// Check total duration of profiles
AssertEquals_LREAL(Expected := 4.0, Actual := ruckig.Trajectory.Duration, DELTA := 1E-8, Message := 'Duration incorrect');

// Check minimum duration
AssertEquals_LREAL(Expected := input.MinDuration, Actual := ruckig.Trajectory.Duration, DELTA := 1E-8, Message := 'Minimum duration not equals duration');

// Check duration for each phase
positionExtrema := ruckig.Trajectory._profiles[0].positionExtrema();
AssertEquals_LREAL(0.0, positionExtrema.Tmax, 1E-9, message:='Profile[0] Tmax incorrect');
AssertEquals_LREAL(61.37396011937787, positionExtrema.Maximum, 1E-9, message:='Profile[0] maximum incorrect');
AssertEquals_LREAL(4.0, positionExtrema.Tmin, 1E-9, message:='Profile[0] Tmin incorrect');
AssertEquals_LREAL(-932.2714554581783, positionExtrema.Minimum, 1E-9, message:='Profile[0] minimum incorrect');

positionExtrema := ruckig.Trajectory._profiles[1].positionExtrema();
AssertEquals_LREAL(4.0, positionExtrema.Tmax, 1E-9, message:='Profile[1] Tmax incorrect');
AssertEquals_LREAL(3356.191464991089, positionExtrema.Maximum, 1E-9, message:='Profile[1] maximum incorrect');
AssertEquals_LREAL(0.10412338784096734, positionExtrema.Tmin, 1E-9, message:='Profile[1] Tmin incorrect');
AssertEquals_LREAL(68.24379604148844, positionExtrema.Minimum, 1E-9, message:='Profile[1] minimum incorrect');

positionExtrema := ruckig.Trajectory._profiles[2].positionExtrema();
AssertEquals_LREAL(0.0, positionExtrema.Tmax, 1E-9, message:='Profile[2] Tmax incorrect');
AssertEquals_LREAL(-8.257039659155268, positionExtrema.Maximum, 1E-9, message:='Profile[2] maximum incorrect');
AssertEquals_LREAL(4.0, positionExtrema.Tmin, 1E-9, message:='Profile[2] Tmin incorrect');
AssertEquals_LREAL(-2142.4383401030323, positionExtrema.Minimum, 1E-9, message:='Profile[2] minimum incorrect');
   

TEST_FINISHED();
END_METHOD

METHOD Test_Trajectory_VelIntrf_HasMinDuration_HasTargetVelocity_HasTargetAcceleration_25
VAR_INST
  ruckig : Struckig.Ruckig(0.001, 0);
  input : Struckig.InputParameter(3) := (
    ControlInterface := ControlInterfaceType.Velocity,
    Synchronization := SynchronizationType.TimeSync,
    MinDuration := 5.0,
    MaxVelocity := [ 2000.0, 2000.0, 2000.0 ],
    MaxAcceleration := [ 20000.0, 20000.0, 20000.0 ],
    MaxJerk := [ 800000.0, 800000.0, 800000.0 ],
    CurrentPosition := [ 99.27158709173054, 51.78630599017913, -82.71240030046118 ],
    CurrentVelocity := [ 617.0096879713556, 556.3356400770322, 654.4714219366203 ],
    CurrentAcceleration := [ 574.9072883020708, 8161.605381343747, 7215.343607485673 ],
    TargetPosition := [ -75.73302485201327, -76.60258111111662, -93.84383456920497 ],
    TargetVelocity := [ -134.5020942775601, 636.5230467842334, -659.8475456020238 ],
    TargetAcceleration := [ -262.53891173287866, -851.053910299499, -307.5361794862756 ]
  );
  
  positionExtrema : Struckig.PositionExtremaDesc;
END_VAR
TEST('Trajectory_VelIntrf_HasMinDuration_HasTargetVelocity_HasTargetAcceleration_25');

ruckig(Input:=input);

// Check total duration of profiles
AssertEquals_LREAL(Expected := 5.0, Actual := ruckig.Trajectory.Duration, DELTA := 1E-8, Message := 'Duration incorrect');

// Check minimum duration
AssertEquals_LREAL(Expected := input.MinDuration, Actual := ruckig.Trajectory.Duration, DELTA := 1E-8, Message := 'Minimum duration not equals duration');

// Check duration for each phase
positionExtrema := ruckig.Trajectory._profiles[0].positionExtrema();
AssertEquals_LREAL(5.0, positionExtrema.Tmax, 1E-9, message:='Profile[0] Tmax incorrect');
AssertEquals_LREAL(2457.793957890017, positionExtrema.Maximum, 1E-9, message:='Profile[0] maximum incorrect');
AssertEquals_LREAL(0.0, positionExtrema.Tmin, 1E-9, message:='Profile[0] Tmin incorrect');
AssertEquals_LREAL(99.27158709173054, positionExtrema.Minimum, 1E-9, message:='Profile[0] minimum incorrect');

positionExtrema := ruckig.Trajectory._profiles[1].positionExtrema();
AssertEquals_LREAL(5.0, positionExtrema.Tmax, 1E-9, message:='Profile[1] Tmax incorrect');
AssertEquals_LREAL(12482.220923700503, positionExtrema.Maximum, 1E-9, message:='Profile[1] maximum incorrect');
AssertEquals_LREAL(0.0, positionExtrema.Tmin, 1E-9, message:='Profile[1] Tmin incorrect');
AssertEquals_LREAL(51.78630599017913, positionExtrema.Minimum, 1E-9, message:='Profile[1] minimum incorrect');

positionExtrema := ruckig.Trajectory._profiles[2].positionExtrema();
AssertEquals_LREAL(5.0, positionExtrema.Tmax, 1E-9, message:='Profile[2] Tmax incorrect');
AssertEquals_LREAL(457.83088712667626, positionExtrema.Maximum, 1E-9, message:='Profile[2] maximum incorrect');
AssertEquals_LREAL(0.0, positionExtrema.Tmin, 1E-9, message:='Profile[2] Tmin incorrect');
AssertEquals_LREAL(-82.71240030046118, positionExtrema.Minimum, 1E-9, message:='Profile[2] minimum incorrect');
   

TEST_FINISHED();
END_METHOD

METHOD Test_Trajectory_VelIntrf_HasMinDuration_HasTargetVelocity_HasTargetAcceleration_26
VAR_INST
  ruckig : Struckig.Ruckig(0.001, 0);
  input : Struckig.InputParameter(3) := (
    ControlInterface := ControlInterfaceType.Velocity,
    Synchronization := SynchronizationType.TimeSync,
    MinDuration := 2.0,
    MaxVelocity := [ 2000.0, 2000.0, 2000.0 ],
    MaxAcceleration := [ 20000.0, 20000.0, 20000.0 ],
    MaxJerk := [ 800000.0, 800000.0, 800000.0 ],
    CurrentPosition := [ 47.83664173753348, -4.090200694219973, 75.62715399288581 ],
    CurrentVelocity := [ -412.71660212910535, -344.97977752529744, -662.3972561668236 ],
    CurrentAcceleration := [ 9700.323608694027, 4925.451680171778, 528.779511900253 ],
    TargetPosition := [ -26.350792724711255, -10.804969468053471, -80.84927076896919 ],
    TargetVelocity := [ -661.2515009925905, -544.0751045990595, 389.8586138148876 ],
    TargetAcceleration := [ -326.74185324603604, 477.02942558038353, -127.6960040536186 ]
  );
  
  positionExtrema : Struckig.PositionExtremaDesc;
END_VAR
TEST('Trajectory_VelIntrf_HasMinDuration_HasTargetVelocity_HasTargetAcceleration_26');

ruckig(Input:=input);

// Check total duration of profiles
AssertEquals_LREAL(Expected := 2.0, Actual := ruckig.Trajectory.Duration, DELTA := 1E-8, Message := 'Duration incorrect');

// Check minimum duration
AssertEquals_LREAL(Expected := input.MinDuration, Actual := ruckig.Trajectory.Duration, DELTA := 1E-8, Message := 'Minimum duration not equals duration');

// Check duration for each phase
positionExtrema := ruckig.Trajectory._profiles[0].positionExtrema();
AssertEquals_LREAL(0.0, positionExtrema.Tmax, 1E-9, message:='Profile[0] Tmax incorrect');
AssertEquals_LREAL(47.83664173753348, positionExtrema.Maximum, 1E-9, message:='Profile[0] maximum incorrect');
AssertEquals_LREAL(2.0, positionExtrema.Tmin, 1E-9, message:='Profile[0] Tmin incorrect');
AssertEquals_LREAL(-965.6623915281051, positionExtrema.Minimum, 1E-9, message:='Profile[0] minimum incorrect');

positionExtrema := ruckig.Trajectory._profiles[1].positionExtrema();
AssertEquals_LREAL(0.0, positionExtrema.Tmax, 1E-9, message:='Profile[1] Tmax incorrect');
AssertEquals_LREAL(-4.090200694219973, positionExtrema.Maximum, 1E-9, message:='Profile[1] maximum incorrect');
AssertEquals_LREAL(2.0, positionExtrema.Tmin, 1E-9, message:='Profile[1] Tmin incorrect');
AssertEquals_LREAL(-877.5597601233831, positionExtrema.Minimum, 1E-9, message:='Profile[1] minimum incorrect');

positionExtrema := ruckig.Trajectory._profiles[2].positionExtrema();
AssertEquals_LREAL(0.0, positionExtrema.Tmax, 1E-9, message:='Profile[2] Tmax incorrect');
AssertEquals_LREAL(75.62715399288581, positionExtrema.Maximum, 1E-9, message:='Profile[2] maximum incorrect');
AssertEquals_LREAL(1.9991825530237812, positionExtrema.Tmin, 1E-9, message:='Profile[2] Tmin incorrect');
AssertEquals_LREAL(-196.96292798248453, positionExtrema.Minimum, 1E-9, message:='Profile[2] minimum incorrect');
   

TEST_FINISHED();
END_METHOD

METHOD Test_Trajectory_VelIntrf_HasMinDuration_HasTargetVelocity_HasTargetAcceleration_33
VAR_INST
  ruckig : Struckig.Ruckig(0.001, 0);
  input : Struckig.InputParameter(3) := (
    ControlInterface := ControlInterfaceType.Velocity,
    Synchronization := SynchronizationType.TimeSync,
    MinDuration := 1.0,
    MaxVelocity := [ 2000.0, 2000.0, 2000.0 ],
    MaxAcceleration := [ 20000.0, 20000.0, 20000.0 ],
    MaxJerk := [ 800000.0, 800000.0, 800000.0 ],
    CurrentPosition := [ -49.2031444482373, -51.45640574706518, 70.88792157601674 ],
    CurrentVelocity := [ -496.32492650532754, -32.672137553484845, 433.6351152131574 ],
    CurrentAcceleration := [ 5796.767034802937, 149.52817879179565, 5479.773632181257 ],
    TargetPosition := [ -60.683308313785076, -77.36542095799315, 35.25281163323578 ],
    TargetVelocity := [ -239.87671609275264, 822.5237555037947, -341.77342454738846 ],
    TargetAcceleration := [ 442.7287565429956, -997.6913770242959, -816.4447449025389 ]
  );
  
  positionExtrema : Struckig.PositionExtremaDesc;
END_VAR
TEST('Trajectory_VelIntrf_HasMinDuration_HasTargetVelocity_HasTargetAcceleration_33');

ruckig(Input:=input);

// Check total duration of profiles
AssertEquals_LREAL(Expected := 1.0, Actual := ruckig.Trajectory.Duration, DELTA := 1E-8, Message := 'Duration incorrect');

// Check minimum duration
AssertEquals_LREAL(Expected := input.MinDuration, Actual := ruckig.Trajectory.Duration, DELTA := 1E-8, Message := 'Minimum duration not equals duration');

// Check duration for each phase
positionExtrema := ruckig.Trajectory._profiles[0].positionExtrema();
AssertEquals_LREAL(0.0, positionExtrema.Tmax, 1E-9, message:='Profile[0] Tmax incorrect');
AssertEquals_LREAL(-49.2031444482373, positionExtrema.Maximum, 1E-9, message:='Profile[0] maximum incorrect');
AssertEquals_LREAL(1.0, positionExtrema.Tmin, 1E-9, message:='Profile[0] Tmin incorrect');
AssertEquals_LREAL(-407.7025966385173, positionExtrema.Minimum, 1E-9, message:='Profile[0] minimum incorrect');

positionExtrema := ruckig.Trajectory._profiles[1].positionExtrema();
AssertEquals_LREAL(1.0, positionExtrema.Tmax, 1E-9, message:='Profile[1] Tmax incorrect');
AssertEquals_LREAL(344.3868574234848, positionExtrema.Maximum, 1E-9, message:='Profile[1] maximum incorrect');
AssertEquals_LREAL(0.000885165723529272, positionExtrema.Tmin, 1E-9, message:='Profile[1] Tmin incorrect');
AssertEquals_LREAL(-51.485174951826146, positionExtrema.Minimum, 1E-9, message:='Profile[1] minimum incorrect');

positionExtrema := ruckig.Trajectory._profiles[2].positionExtrema();
AssertEquals_LREAL(0.9999795141123666, positionExtrema.Tmax, 1E-9, message:='Profile[2] Tmax incorrect');
AssertEquals_LREAL(129.085190687188, positionExtrema.Maximum, 1E-9, message:='Profile[2] maximum incorrect');
AssertEquals_LREAL(0.0, positionExtrema.Tmin, 1E-9, message:='Profile[2] Tmin incorrect');
AssertEquals_LREAL(70.88792157601674, positionExtrema.Minimum, 1E-9, message:='Profile[2] minimum incorrect');
   

TEST_FINISHED();
END_METHOD

METHOD Test_Trajectory_VelIntrf_HasMinDuration_HasTargetVelocity_HasTargetAcceleration_37
VAR_INST
  ruckig : Struckig.Ruckig(0.001, 0);
  input : Struckig.InputParameter(3) := (
    ControlInterface := ControlInterfaceType.Velocity,
    Synchronization := SynchronizationType.TimeSync,
    MinDuration := 2.0,
    MaxVelocity := [ 2000.0, 2000.0, 2000.0 ],
    MaxAcceleration := [ 20000.0, 20000.0, 20000.0 ],
    MaxJerk := [ 800000.0, 800000.0, 800000.0 ],
    CurrentPosition := [ -12.004712599902348, 73.67282675877655, -52.349457595484836 ],
    CurrentVelocity := [ 292.20783385007076, -778.1307817801523, -64.33328614652999 ],
    CurrentAcceleration := [ 245.56834991156393, 4188.319168784961, -3762.4320312456057 ],
    TargetPosition := [ 82.49345668673473, 58.903290717842765, 34.45715254310531 ],
    TargetVelocity := [ -333.20598063149066, 685.2693740134762, 482.0796900333503 ],
    TargetAcceleration := [ 240.05556433564402, -666.6421184257438, -752.3384651343332 ]
  );
  
  positionExtrema : Struckig.PositionExtremaDesc;
END_VAR
TEST('Trajectory_VelIntrf_HasMinDuration_HasTargetVelocity_HasTargetAcceleration_37');

ruckig(Input:=input);

// Check total duration of profiles
AssertEquals_LREAL(Expected := 2.0, Actual := ruckig.Trajectory.Duration, DELTA := 1E-8, Message := 'Duration incorrect');

// Check minimum duration
AssertEquals_LREAL(Expected := input.MinDuration, Actual := ruckig.Trajectory.Duration, DELTA := 1E-8, Message := 'Minimum duration not equals duration');

// Check duration for each phase
positionExtrema := ruckig.Trajectory._profiles[0].positionExtrema();
AssertEquals_LREAL(0.0006980853396357632, positionExtrema.Tmax, 1E-9, message:='Profile[0] Tmax incorrect');
AssertEquals_LREAL(-11.80071211848046, positionExtrema.Maximum, 1E-9, message:='Profile[0] maximum incorrect');
AssertEquals_LREAL(2.0, positionExtrema.Tmin, 1E-9, message:='Profile[0] Tmin incorrect');
AssertEquals_LREAL(-52.999031310760635, positionExtrema.Minimum, 1E-9, message:='Profile[0] minimum incorrect');

positionExtrema := ruckig.Trajectory._profiles[1].positionExtrema();
AssertEquals_LREAL(2.0, positionExtrema.Tmax, 1E-9, message:='Profile[1] Tmax incorrect');
AssertEquals_LREAL(1703.4819483796325, positionExtrema.Maximum, 1E-9, message:='Profile[1] maximum incorrect');
AssertEquals_LREAL(0.207432051719431, positionExtrema.Tmin, 1E-9, message:='Profile[1] Tmin incorrect');
AssertEquals_LREAL(-3.8974776087497673, positionExtrema.Minimum, 1E-9, message:='Profile[1] minimum incorrect');

positionExtrema := ruckig.Trajectory._profiles[2].positionExtrema();
AssertEquals_LREAL(2.0, positionExtrema.Tmax, 1E-9, message:='Profile[2] Tmax incorrect');
AssertEquals_LREAL(355.8717476818793, positionExtrema.Maximum, 1E-9, message:='Profile[2] maximum incorrect');
AssertEquals_LREAL(0.005051342367393055, positionExtrema.Tmin, 1E-9, message:='Profile[2] Tmin incorrect');
AssertEquals_LREAL(-52.70524288915402, positionExtrema.Minimum, 1E-9, message:='Profile[2] minimum incorrect');
   

TEST_FINISHED();
END_METHOD

METHOD Test_Trajectory_VelIntrf_HasMinDuration_HasTargetVelocity_HasTargetAcceleration_40
VAR_INST
  ruckig : Struckig.Ruckig(0.001, 0);
  input : Struckig.InputParameter(3) := (
    ControlInterface := ControlInterfaceType.Velocity,
    Synchronization := SynchronizationType.TimeSync,
    MinDuration := 4.0,
    MaxVelocity := [ 2000.0, 2000.0, 2000.0 ],
    MaxAcceleration := [ 20000.0, 20000.0, 20000.0 ],
    MaxJerk := [ 800000.0, 800000.0, 800000.0 ],
    CurrentPosition := [ -76.42035041184897, -68.81061285502989, 60.15861595713818 ],
    CurrentVelocity := [ 424.8413928919874, 178.96533202855449, 765.6862190691088 ],
    CurrentAcceleration := [ 1338.04438518401, 3559.2301009959247, -1023.1564895528609 ],
    TargetPosition := [ -17.943807189703136, 56.757291906819944, -0.6309720814246589 ],
    TargetVelocity := [ -763.7685723303848, 641.2936977777251, -718.0886986858688 ],
    TargetAcceleration := [ 498.71648374610845, -601.18528422182, -73.467606210815 ]
  );
  
  positionExtrema : Struckig.PositionExtremaDesc;
END_VAR
TEST('Trajectory_VelIntrf_HasMinDuration_HasTargetVelocity_HasTargetAcceleration_40');

ruckig(Input:=input);

// Check total duration of profiles
AssertEquals_LREAL(Expected := 4.0, Actual := ruckig.Trajectory.Duration, DELTA := 1E-8, Message := 'Duration incorrect');

// Check minimum duration
AssertEquals_LREAL(Expected := input.MinDuration, Actual := ruckig.Trajectory.Duration, DELTA := 1E-8, Message := 'Minimum duration not equals duration');

// Check duration for each phase
positionExtrema := ruckig.Trajectory._profiles[0].positionExtrema();
AssertEquals_LREAL(0.0020446425392176273, positionExtrema.Tmax, 1E-9, message:='Profile[0] Tmax incorrect');
AssertEquals_LREAL(-75.5500444389785, positionExtrema.Maximum, 1E-9, message:='Profile[0] maximum incorrect');
AssertEquals_LREAL(4.0, positionExtrema.Tmin, 1E-9, message:='Profile[0] Tmin incorrect');
AssertEquals_LREAL(-751.7240555499565, positionExtrema.Minimum, 1E-9, message:='Profile[0] minimum incorrect');

positionExtrema := ruckig.Trajectory._profiles[1].positionExtrema();
AssertEquals_LREAL(4.0, positionExtrema.Tmax, 1E-9, message:='Profile[1] Tmax incorrect');
AssertEquals_LREAL(5988.6562563663865, positionExtrema.Maximum, 1E-9, message:='Profile[1] maximum incorrect');
AssertEquals_LREAL(0.0, positionExtrema.Tmin, 1E-9, message:='Profile[1] Tmin incorrect');
AssertEquals_LREAL(-68.81061285502989, positionExtrema.Minimum, 1E-9, message:='Profile[1] minimum incorrect');

positionExtrema := ruckig.Trajectory._profiles[2].positionExtrema();
AssertEquals_LREAL(0.897558808059484, positionExtrema.Tmax, 1E-9, message:='Profile[2] Tmax incorrect');
AssertEquals_LREAL(380.9463968009695, positionExtrema.Maximum, 1E-9, message:='Profile[2] maximum incorrect');
AssertEquals_LREAL(4.0, positionExtrema.Tmin, 1E-9, message:='Profile[2] Tmin incorrect');
AssertEquals_LREAL(-1230.5349501304436, positionExtrema.Minimum, 1E-9, message:='Profile[2] minimum incorrect');
   

TEST_FINISHED();
END_METHOD

METHOD Test_Trajectory_VelIntrf_HasMinDuration_HasTargetVelocity_HasTargetAcceleration_9
VAR_INST
  ruckig : Struckig.Ruckig(0.001, 0);
  input : Struckig.InputParameter(3) := (
    ControlInterface := ControlInterfaceType.Velocity,
    Synchronization := SynchronizationType.TimeSync,
    MinDuration := 7.0,
    MaxVelocity := [ 2000.0, 2000.0, 2000.0 ],
    MaxAcceleration := [ 20000.0, 20000.0, 20000.0 ],
    MaxJerk := [ 800000.0, 800000.0, 800000.0 ],
    CurrentPosition := [ 65.33675034249944, 20.471874067999465, 17.7936900678952 ],
    CurrentVelocity := [ 251.51375561632767, -883.355945316876, 592.220566480973 ],
    CurrentAcceleration := [ 9181.774579926536, -9976.3302467699, 2745.115542495065 ],
    TargetPosition := [ -63.4605755257718, 16.3093879856457, -25.6649619333392 ],
    TargetVelocity := [ 614.4494968030804, -34.17434532431503, 533.9879492839282 ],
    TargetAcceleration := [ -792.1476751145624, 673.4644110073796, -240.28714730173158 ]
  );
  
  positionExtrema : Struckig.PositionExtremaDesc;
END_VAR
TEST('Trajectory_VelIntrf_HasMinDuration_HasTargetVelocity_HasTargetAcceleration_9');

ruckig(Input:=input);

// Check total duration of profiles
AssertEquals_LREAL(Expected := 7.0, Actual := ruckig.Trajectory.Duration, DELTA := 1E-8, Message := 'Duration incorrect');

// Check minimum duration
AssertEquals_LREAL(Expected := input.MinDuration, Actual := ruckig.Trajectory.Duration, DELTA := 1E-8, Message := 'Minimum duration not equals duration');

// Check duration for each phase
positionExtrema := ruckig.Trajectory._profiles[0].positionExtrema();
AssertEquals_LREAL(7.0, positionExtrema.Tmax, 1E-9, message:='Profile[0] Tmax incorrect');
AssertEquals_LREAL(21441.07705236427, positionExtrema.Maximum, 1E-9, message:='Profile[0] maximum incorrect');
AssertEquals_LREAL(0.0, positionExtrema.Tmin, 1E-9, message:='Profile[0] Tmin incorrect');
AssertEquals_LREAL(65.33675034249944, positionExtrema.Minimum, 1E-9, message:='Profile[0] minimum incorrect');

positionExtrema := ruckig.Trajectory._profiles[1].positionExtrema();
AssertEquals_LREAL(0.0, positionExtrema.Tmax, 1E-9, message:='Profile[1] Tmax incorrect');
AssertEquals_LREAL(20.471874067999465, positionExtrema.Maximum, 1E-9, message:='Profile[1] maximum incorrect');
AssertEquals_LREAL(7.0, positionExtrema.Tmin, 1E-9, message:='Profile[1] Tmin incorrect');
AssertEquals_LREAL(-15783.474903608412, positionExtrema.Minimum, 1E-9, message:='Profile[1] minimum incorrect');

positionExtrema := ruckig.Trajectory._profiles[2].positionExtrema();
AssertEquals_LREAL(7.0, positionExtrema.Tmax, 1E-9, message:='Profile[2] Tmax incorrect');
AssertEquals_LREAL(9053.9566289456, positionExtrema.Maximum, 1E-9, message:='Profile[2] maximum incorrect');
AssertEquals_LREAL(0.0, positionExtrema.Tmin, 1E-9, message:='Profile[2] Tmin incorrect');
AssertEquals_LREAL(17.7936900678952, positionExtrema.Minimum, 1E-9, message:='Profile[2] minimum incorrect');
   

TEST_FINISHED();
END_METHOD

END_FUNCTION_BLOCK

(* stored: Version 1.1.0.1, ProductVersion 3.1.4024.9
   POU VelocityInterfaceTest: Id {8a002d40-1b8b-4a36-917f-04dd149a7db3}, SpecialFunc None
   Method Test_Trajectory_VelIntrf_HasMinDuration_11: Id {99a7cccb-ff59-4929-aa01-691b630484c7}
   Method Test_Trajectory_VelIntrf_HasMinDuration_13: Id {0ef65899-97d4-4574-84d9-398de273b398}
   Method Test_Trajectory_VelIntrf_HasMinDuration_16: Id {a955ef3b-d470-4da7-833e-0ecec8a02a2d}
   Method Test_Trajectory_VelIntrf_HasMinDuration_18: Id {af1fba8f-a368-414e-a553-dadddefe26ef}
   Method Test_Trajectory_VelIntrf_HasMinDuration_27: Id {a5d4f584-6624-45c8-aa14-27f80ba83a5d}
   Method Test_Trajectory_VelIntrf_HasMinDuration_3: Id {8dc05fdc-7087-4b57-87d4-f2e05b72a055}
   Method Test_Trajectory_VelIntrf_HasMinDuration_30: Id {8efc570b-dfc1-4d70-9020-2c6a5f86cc10}
   Method Test_Trajectory_VelIntrf_HasMinDuration_32: Id {3c8c571f-c69b-418c-aa4d-238f8659b13b}
   Method Test_Trajectory_VelIntrf_HasMinDuration_34: Id {de8f6ecb-1872-45a0-84ee-604aa3b7ed93}
   Method Test_Trajectory_VelIntrf_HasMinDuration_36: Id {b1bebb7e-2df7-496a-b2c5-31d9f60b246d}
   Method Test_Trajectory_VelIntrf_HasMinDuration_38: Id {0ce8f503-3dc7-45b5-9ceb-668e474ba9a2}
   Method Test_Trajectory_VelIntrf_HasMinDuration_39: Id {9da3f16c-d146-4570-856f-0d8ba7b09a4f}
   Method Test_Trajectory_VelIntrf_HasMinDuration_4: Id {749a1204-c253-40b6-af28-96c08426d3ae}
   Method Test_Trajectory_VelIntrf_HasMinDuration_6: Id {a214fb44-210a-4996-9682-8d59b300b757}
   Method Test_Trajectory_VelIntrf_HasMinDuration_8: Id {6db2d1ba-a4dc-4f54-9510-7e3b8fd834db}
   Method Test_Trajectory_VelIntrf_HasMinDuration_HasTargetAcceleration_12: Id {0221d664-422c-4732-b9fb-c40d7f69f6ad}
   Method Test_Trajectory_VelIntrf_HasMinDuration_HasTargetAcceleration_14: Id {08de52b7-af44-4bc1-bbf1-54612e29fccd}
   Method Test_Trajectory_VelIntrf_HasMinDuration_HasTargetAcceleration_15: Id {69e6a053-1957-4573-8682-9a2718d43b24}
   Method Test_Trajectory_VelIntrf_HasMinDuration_HasTargetAcceleration_2: Id {c1d284a6-5e38-46c5-b740-426065c57fc4}
   Method Test_Trajectory_VelIntrf_HasMinDuration_HasTargetAcceleration_24: Id {5263eb97-44d9-44ac-8f39-76ea9cbec470}
   Method Test_Trajectory_VelIntrf_HasMinDuration_HasTargetAcceleration_28: Id {2e790798-1293-4293-8eb2-628a9c0e1a21}
   Method Test_Trajectory_VelIntrf_HasMinDuration_HasTargetVelocity_10: Id {f41d6d28-c33d-4b2f-b6ee-1e653253a105}
   Method Test_Trajectory_VelIntrf_HasMinDuration_HasTargetVelocity_29: Id {5bad9645-97b6-4927-b3eb-8f87324b1ece}
   Method Test_Trajectory_VelIntrf_HasMinDuration_HasTargetVelocity_31: Id {91e39518-d20f-4466-b934-2a532a163bd6}
   Method Test_Trajectory_VelIntrf_HasMinDuration_HasTargetVelocity_35: Id {bc69f65e-3d82-488c-9a8d-925025f7583a}
   Method Test_Trajectory_VelIntrf_HasMinDuration_HasTargetVelocity_5: Id {2f753f46-c298-4c4a-921d-972d6cb39a4e}
   Method Test_Trajectory_VelIntrf_HasMinDuration_HasTargetVelocity_7: Id {84d212dd-be99-4296-81ee-d752aa16c4b5}
   Method Test_Trajectory_VelIntrf_HasMinDuration_HasTargetVelocity_HasTargetAcceleration_1: Id {a4116616-8c2a-4850-9bbb-663da589817a}
   Method Test_Trajectory_VelIntrf_HasMinDuration_HasTargetVelocity_HasTargetAcceleration_17: Id {d93492c0-13b3-4877-9d56-8e6aec3f5202}
   Method Test_Trajectory_VelIntrf_HasMinDuration_HasTargetVelocity_HasTargetAcceleration_19: Id {aa9f23a5-a5e3-4b63-b9ab-497338e2669a}
   Method Test_Trajectory_VelIntrf_HasMinDuration_HasTargetVelocity_HasTargetAcceleration_20: Id {bf0ead00-4904-4fd7-8f11-e8ad3253a125}
   Method Test_Trajectory_VelIntrf_HasMinDuration_HasTargetVelocity_HasTargetAcceleration_21: Id {b2dca3c6-72fe-4411-866c-cbce9aed8712}
   Method Test_Trajectory_VelIntrf_HasMinDuration_HasTargetVelocity_HasTargetAcceleration_22: Id {ebcb322a-b7c5-439c-b8d9-f4439cbd7cad}
   Method Test_Trajectory_VelIntrf_HasMinDuration_HasTargetVelocity_HasTargetAcceleration_23: Id {234c021c-2393-4616-a082-6a6abf8c02ce}
   Method Test_Trajectory_VelIntrf_HasMinDuration_HasTargetVelocity_HasTargetAcceleration_25: Id {b2c92848-2a1e-4418-9790-582ff37301e1}
   Method Test_Trajectory_VelIntrf_HasMinDuration_HasTargetVelocity_HasTargetAcceleration_26: Id {bd58012d-cbc2-496e-b5dd-fbcc2f4f586b}
   Method Test_Trajectory_VelIntrf_HasMinDuration_HasTargetVelocity_HasTargetAcceleration_33: Id {d4861a2a-3b67-4d84-87c0-60579366f579}
   Method Test_Trajectory_VelIntrf_HasMinDuration_HasTargetVelocity_HasTargetAcceleration_37: Id {4dd617ac-2f3f-49f6-b627-eaf3e752ec4e}
   Method Test_Trajectory_VelIntrf_HasMinDuration_HasTargetVelocity_HasTargetAcceleration_40: Id {ecd1b891-bba9-490e-bee4-6542e0d38de6}
   Method Test_Trajectory_VelIntrf_HasMinDuration_HasTargetVelocity_HasTargetAcceleration_9: Id {13f98850-97b9-4f5f-8320-4caa648fee04} *)
